# EPICS substitutions: dxp/branches/R3-0-branch/iocBoot/iocXMAP/16element.substitutions
file "$(DXP)/dxpApp/Db/dxpMED.template"
{
pattern
{P,           MCAALL,    INP          }
{dxpXMAP: mcaAll, "@asyn(DXP1,16)"}
}

file "$(MCA)/mcaApp/Db/simple_mca.db"
{
pattern
{       P,      M,       DTYP,               INP,  PREC,    CHANS}
{dxpXMAP:,   mca1,  "asynMCA",   "@asyn(DXP1,0)",     2,     2048}
{dxpXMAP:,   mca2,  "asynMCA",   "@asyn(DXP1,1)",     2,     2048}
{dxpXMAP:,   mca3,  "asynMCA",   "@asyn(DXP1,2)",     2,     2048}
{dxpXMAP:,   mca4,  "asynMCA",   "@asyn(DXP1,3)",     2,     2048}
{dxpXMAP:,   mca5,  "asynMCA",   "@asyn(DXP1,4)",     2,     2048}
{dxpXMAP:,   mca6,  "asynMCA",   "@asyn(DXP1,5)",     2,     2048}
{dxpXMAP:,   mca7,  "asynMCA",   "@asyn(DXP1,6)",     2,     2048}
{dxpXMAP:,   mca8,  "asynMCA",   "@asyn(DXP1,7)",     2,     2048}
{dxpXMAP:,   mca9,  "asynMCA",   "@asyn(DXP1,8)",     2,     2048}
{dxpXMAP:,   mca10, "asynMCA",   "@asyn(DXP1,9)",     2,     2048}
{dxpXMAP:,   mca11, "asynMCA",   "@asyn(DXP1,10)",    2,     2048}
{dxpXMAP:,   mca12, "asynMCA",   "@asyn(DXP1,11)",    2,     2048}
{dxpXMAP:,   mca13, "asynMCA",   "@asyn(DXP1,12)",    2,     2048}
{dxpXMAP:,   mca14, "asynMCA",   "@asyn(DXP1,13)",    2,     2048}
{dxpXMAP:,   mca15, "asynMCA",   "@asyn(DXP1,14)",    2,     2048}
{dxpXMAP:,   mca16, "asynMCA",   "@asyn(DXP1,15)",    2,     2048}
{dxpXMAP:,  mcaAll, "asynMCA",   "@asyn(DXP1,-1)",    2,     2048}
}

# DXP records
file "$(DXP)/dxpApp/Db/dxp.template"
{
pattern
{      P,        R,    PINI,  PORT,   ADDR,    TIMEOUT}
{dxpXMAP:,    dxp1:,    YES,  DXP1,      0,         1}
{dxpXMAP:,    dxp2:,    YES,  DXP1,      1,         1}
{dxpXMAP:,    dxp3:,    YES,  DXP1,      2,         1}
{dxpXMAP:,    dxp4:,    YES,  DXP1,      3,         1}
{dxpXMAP:,    dxp5:,    YES,  DXP1,      4,         1}
{dxpXMAP:,    dxp6:,    YES,  DXP1,      5,         1}
{dxpXMAP:,    dxp7:,    YES,  DXP1,      6,         1}
{dxpXMAP:,    dxp8:,    YES,  DXP1,      7,         1}
{dxpXMAP:,    dxp9:,    YES,  DXP1,      8,         1}
{dxpXMAP:,   dxp10:,    YES,  DXP1,      9,         1}
{dxpXMAP:,   dxp11:,    YES,  DXP1,     10,         1}
{dxpXMAP:,   dxp12:,    YES,  DXP1,     11,         1}
{dxpXMAP:,   dxp13:,    YES,  DXP1,     12,         1}
{dxpXMAP:,   dxp14:,    YES,  DXP1,     13,         1}
{dxpXMAP:,   dxp15:,    YES,  DXP1,     14,         1}
{dxpXMAP:,   dxp16:,    YES,  DXP1,     15,         1}
#{dxpXMAP:  dxpAll:,     NO,  DXP1,     16,         1}
}
